// TIA Portal V19 export
DATA_BLOCK "iDB_FlatnessCtrlRecordLRobot"   // DB711
{ DB_Accessible_From_OPC_UA := 'FALSE' }
// stored: AutoNumber false, DBAccessibleFromOPCUA false, DBAccessibleFromWebserver false, InstanceOfName FB71_FlatnessCtrlRecord, InstanceOfType FB
"FB71_FlatnessCtrlRecord"
   // VAR_OUTPUT
   //    uiRecordMax { ExternalAccessible := 'False'; ExternalVisible := 'False'; ExternalWritable := 'False'} : UInt;
   //    uiRecordMin { ExternalAccessible := 'False'; ExternalVisible := 'False'; ExternalWritable := 'False'} : UInt;
   //    DisplayFlatRecData { ExternalAccessible := 'False'; ExternalVisible := 'False'; ExternalWritable := 'False'} : "stFlatnessCtrlRecord";
   // END_VAR
   // VAR_IN_OUT
   //    xEraseAllData { ExternalAccessible := 'False'; ExternalVisible := 'False'; ExternalWritable := 'False'} : Bool;
   //    xDisplayNextRecord { ExternalAccessible := 'False'; ExternalVisible := 'False'; ExternalWritable := 'False'} : Bool;
   //    xDisplayPrevRecord { ExternalAccessible := 'False'; ExternalVisible := 'False'; ExternalWritable := 'False'} : Bool;
   //    uiDisplayCurentRecord { ExternalAccessible := 'False'; ExternalVisible := 'False'; ExternalWritable := 'False'} : UInt;
   //    uiNumberOfRecords { ExternalAccessible := 'False'; ExternalVisible := 'False'; ExternalWritable := 'False'} : UInt;
   //    stFlatnessdata : "stFlatnessData";
   //    aFlatnessData : Array[*] of "stFlatnessCtrlRecord";
   // END_VAR
   // VAR
   //    sdiMaxRecord { ExternalAccessible := 'False'; ExternalVisible := 'False'; ExternalWritable := 'False'} : DInt;
   //    siCounter { ExternalAccessible := 'False'; ExternalVisible := 'False'; ExternalWritable := 'False'} : Int;
   //    suiMemDisplayCurentReccord { ExternalAccessible := 'False'; ExternalVisible := 'False'; ExternalWritable := 'False'} : UInt;
   // END_VAR
BEGIN
END_DATA_BLOCK
